// TIA Portal V19 export
TYPE "udt_FsParameter"
   STRUCT
      WorkMode : UInt;
      Positions : Struct
         HomePosition : LReal;
         WorkEnablePosition : LReal;
         ReturnEnablePosition : LReal;
         StillCutPosition : LReal := 1000.0;
      END_STRUCT;
      ToolCycleTime : LReal := 1.0;
      FollowingErrorWindow : LReal := 0.1;
      DwellTimeErrorWindow : Time := T#100ms;
      ErrorTimeout : Time := T#1s;
      BladeDetachValue : LReal;
      BladeDetachVelocity : LReal;
      SyncDinamics : Struct
         Acceleration : LReal;
         Jerk : LReal;
         ReturnVelocity : LReal;
         StartAdvanceSpace : LReal := 50.0;
         SyncLag : LReal := 10.0;
         ExtraSpeed : Real := 1.0;
      END_STRUCT;
   END_STRUCT;
END_TYPE
